INTERFACE ITF_BaseHMIGroupElement_Command EXTENDS ITF_BaseHMIControlElement_Command

END_INTERFACE

(* stored: Version 1.1.0.1
   Itf ITF_BaseHMIGroupElement_Command: Id {8272aa8f-99f8-002f-1ba5-66436cdc2b46} *)
